Staubli VAL3: debugMsg.pgx

public program debugMsg(num x_nDebug (dimensions=1))
begin
  //-----------------------------------------------------------------------
  //Header begin
  //Description of program
  //  Enable/Disable debug : displays error messages when an error occurs.
  //
  //Input parameters
  //  num x_nDebug : enable/disable errors messages
  //    possible values : 0 -> Disable errors messages
  //                      1 -> Enable Socket errors messages
  //                      2 -> Enable Programs errors messages
  //                      3 -> Enable Socket/Programs errors messages
  //
  //Examples
  //  call debugMsg(1)
  //
  //History
  //  Creation : 19-05-08 - f.Rob
  //Header end
  //-----------------------------------------------------------------------

  switch x_nDebug
    //Disable errors messages
    case 0
      bDebugProgram=bDebugSocket=false
    break
    //Enable Socket errors messages
    case 1
      bDebugProgram=true
      bDebugSocket=false
    break
    //Enable Programs errors messages
    case 2
      bDebugProgram=false
      bDebugSocket=true
    break
    //Enable Socket/Programs errors messages
    case 3
      bDebugProgram=bDebugSocket=true
    break
  endSwitch
end
